Yaskawa INFORM job: KRIS_OTHER_WELDS.JBI

/JOB
//NAME KRIS_OTHER_WELDS
//POS
///NPOS 370,370,370,14,0,0
///TOOL 0
///POSTYPE PULSE
///PULSE
C00000=-36471,-76527,-106813,19264,71481,77238
C00001=-104392,-45604,-45068,-41730,67848,-43971
C00002=-102772,-23592,-15673,-48581,65359,-41958
C00003=-103105,-4521,-1193,-48225,65783,-42370
C00004=-103550,-365,5452,-48799,64222,-41754
C00005=-103550,625,8518,-49296,63299,-41230
C00006=-103550,355,7706,-49163,63541,-41368
C00007=-102300,1028,8270,-49380,64218,-41057
C00008=-102134,1217,8640,-49454,64220,-40967
C00009=-102487,1102,8722,-49434,63955,-41010
C00010=-101792,827,6993,-49227,64947,-41190
C00011=-100819,-958,-818,-48185,68095,-42388
C00012=-74228,-100728,-57385,-53918,72446,-30220
C00013=-60504,-146661,-111893,-16693,92041,63510
C00014=-81002,-144165,-111893,-31958,74905,63510
C00015=-99609,-128801,-101652,-29194,69226,57515
C00016=-99609,-127984,-100239,-29275,68831,57620
C00017=-99609,-128289,-100766,-29244,68978,57581
C00018=-102150,-129321,-101059,-28822,67791,56859
C00019=-99944,-132310,-102446,-29373,67957,57721
C00020=-94854,-157221,-110079,-32013,62771,61374
C00021=-94854,-157221,-110079,-32013,62771,61374
C00022=-150575,-180894,-113467,20602,37776,-7473
C00023=-131435,-154210,-106652,7413,43941,3112
C00024=-131414,-154056,-106648,7392,44016,3129
C00025=-131048,-150684,-105922,7028,45259,3400
C00026=-131414,-154056,-106648,7392,44016,3129
C00027=-178670,-106537,-94441,32173,86364,-27351
C00028=-174579,-86120,-85943,32864,94727,-28981
C00029=-173469,-85635,-85233,32803,94141,-28710
C00030=-173469,-85539,-84108,32766,93596,-28870
C00031=-173084,-86046,-85408,32780,93905,-28625
C00032=-171779,-87936,-86208,32689,92999,-28371
C00033=-172551,-86827,-85740,32743,93534,-28522
C00034=-185237,-110424,-94728,32531,92831,-33795
C00035=-185237,-110424,-94728,32531,92831,-33795
C00036=-134012,-175619,-118342,-2096,46955,2797
C00037=-133371,-126486,-107062,-2327,67886,2658
C00038=-134292,-123400,-104700,-2048,67993,2322
C00039=-134292,-122480,-102592,-2060,67168,2335
C00040=-134292,-122828,-103379,-2055,67474,2331
C00041=-133740,-117277,-101631,-2195,69264,2498
C00042=-134292,-122828,-103379,-2055,67474,2331
C00043=-145565,-124760,-104669,1363,67226,-1769
C00044=-155916,-134756,-102618,15305,54723,-11432
C00045=-154931,-135462,-102806,14939,54301,-11078
C00046=-159722,-139649,-104449,17130,54142,-13140
C00047=-121501,-151260,-116369,-16790,67529,22254
C00048=-84851,-125920,-106326,-14509,72614,18670
C00049=-87302,-113526,-101119,-13757,75261,17475
C00050=-88050,-112106,-100360,-13572,75391,17193
C00051=-88050,-111725,-99039,-13608,74790,17261
C00052=-88050,-111984,-99928,-13584,75193,17215
C00053=-88832,-108808,-98834,-13352,75998,16846
C00054=-87807,-112947,-100252,-13656,74947,17329
C00055=-92070,-142291,-103311,-16392,49176,14760
C00056=-92668,-139554,-102636,-15878,50013,14349
C00057=-91121,-138706,-102421,-16531,50612,14939
C00058=-93561,-140381,-102567,-15560,49394,14049
C00059=-69173,-195704,-118009,-34153,38892,29324
C00060=-69173,-195704,-118009,-34153,38892,29324
C00061=-107696,-37154,-67359,-5229,84713,5863
C00062=-116742,-32674,-55171,-12076,80004,1616
C00063=-117154,-30403,-53709,-11929,80206,1458
C00064=-117154,-30689,-52627,-11956,79411,1536
C00065=-117154,-30552,-53163,-11943,79803,1497
C00066=-108517,-16990,-43540,-23191,88993,13455
C00067=-109765,-14828,-41918,-22897,88763,13064
C00068=-109347,-17906,-44920,-22997,89117,13141
C00069=-106896,-6499,-37008,-27511,96493,19470
C00070=-107863,-6880,-37313,-27352,96184,19193
C00071=-104662,-5505,-36210,-27871,97208,20107
C00072=-93389,-55640,-71668,-19302,82770,9184
C00073=-93389,-55640,-71668,-19302,92834,-78584
C00074=-111754,-46764,-69921,-16160,92456,-84768
C00075=-113010,-47490,-70150,-15902,91999,-85126
C00076=-113010,-47824,-69220,-15892,91281,-85034
C00077=-113010,-47731,-69491,-15895,91487,-85061
C00078=-112902,-49890,-70751,-15912,91185,-84985
C00079=-100788,-44242,-62951,-32464,93570,-83345
C00080=-95750,-41506,-57227,-39958,94516,-82624
C00081=-97351,-42547,-57870,-39748,93692,-82997
C00082=-107713,-44703,-69881,-16984,94226,-83661
C00083=-110462,-17925,-52010,-16025,110800,-86473
C00084=-113105,-11726,-45581,-15485,114570,-87767
C00085=-116727,-11513,-45414,-15662,113935,-88992
C00086=-102039,-2481,-42089,-15122,118996,-84328
C00087=-102039,-2481,-42089,-15122,100704,14672
C00088=-117847,-25402,-50017,-12117,83012,11069
C00089=-117859,-24620,-49869,-12107,83315,11036
C00090=-117859,-24721,-49537,-12111,83065,11060
C00091=-117448,-24507,-49386,-12236,83141,11189
C00092=-109902,-9247,-38011,-19141,88596,18895
C00093=-104609,19012,-13716,-27585,102398,34238
C00094=-104836,21780,-11197,-27552,102213,34199
C00095=-98934,25941,-685,-39115,101412,35075
C00096=-91600,14785,-13342,-39748,106246,36411
C00097=-47111,-89064,-83881,-31350,116876,52529
C00098=-81588,-140072,-114826,-15376,71241,20037
C00099=-97769,-116268,-100554,-7249,70146,8698
C00100=-93709,-113858,-99760,-8341,71283,10082
C00101=-110362,-115244,-100357,6076,70211,-7492
C00102=-124823,-97243,-93907,17727,83078,-24095
C00103=-122674,-104476,-96562,17426,80631,-23684
C00104=-131812,-116317,-102091,19024,80117,-27039
C00105=-131812,-116317,-102091,19024,80117,-27039
C00106=-106372,-151670,-115941,-1479,61909,1124
C00107=-97402,-154853,-108420,-9880,47553,8329
C00108=-91237,-150897,-107478,-16251,51513,16477
C00109=-91228,-148864,-107179,-20465,55021,21052
C00110=-78071,-160284,-116606,-19433,65818,26969
C00111=-78071,-160284,-116606,-19433,65818,26969
C00112=-90794,-133617,-109168,-16116,71767,21274
C00113=-91693,-124585,-104857,-15775,73503,20713
C00114=-94506,-128481,-105877,-15295,71639,19928
C00115=-115362,-143961,-110168,-10698,63087,13119
C00116=-118733,-159504,-110501,-11315,48800,13248
C00117=-120726,-159269,-110393,-10449,48589,12395
C00118=-145117,-154970,-109769,815,48979,1768
C00119=-160284,-149983,-108729,14151,53864,-11283
C00120=-160335,-149941,-108719,14167,53888,-11301
C00121=-182605,-105442,-95794,27625,86766,-32303
C00122=-182041,-70442,-81142,28906,106085,-40460
C00123=-180373,-64217,-77967,29369,107732,-40648
C00124=-198406,-78013,-87317,27723,112552,-46613
C00125=-172769,-133105,-108161,-8035,62165,26522
C00126=-178553,-109735,-99654,4570,64842,24680
C00127=-178553,-100066,-94046,4517,66355,24740
C00128=-175583,-95072,-92228,3296,67653,25861
C00129=-192352,-138021,-108691,10814,57252,18824
C00130=-195651,-141887,-109704,12316,56387,17389
C00131=-195651,-141887,-109704,12316,56387,17389
C00132=-147222,-76033,-86464,-7641,74662,35625
C00133=-144580,-61393,-75556,-8586,75722,36452
C00134=-156265,-37930,-66612,3030,87434,69848
C00135=-155034,-33755,-60965,2668,86065,70206
C00136=-154458,-32798,-60008,2135,86746,70342
C00137=-155825,-31413,-58479,2524,86554,69904
C00138=-162790,-57725,-64353,16754,59169,66258
C00139=-162790,-57725,-64353,16754,59169,66258
C00140=-155825,-31413,-58479,2524,86554,69904
C00141=-155825,-31413,-58479,2524,86554,69904
C00142=-162790,-57725,-64353,16754,59169,66258
C00143=-165729,-66356,-73131,18164,60713,65340
C00144=-165729,-63659,-85226,16965,69151,66660
C00145=-19938,-154159,-115231,23119,85461,7967
C00146=-13636,-159467,-113845,12203,49637,17715
C00147=-116484,-130017,-129030,11526,91164,19547
C00148=-116484,-130017,-129030,11526,91164,19547
C00149=-101509,-111741,-97351,-2474,75173,11228
C00150=-109604,-105261,-90247,-737,73969,8417
C00151=-109604,-104665,-88539,-738,73224,8421
C00152=-109604,-104936,-89303,-737,73555,8419
C00153=-110002,-100393,-87649,-645,74866,8273
C00154=-109618,-105123,-90216,-732,74019,8412
C00155=-74185,-80593,-80392,-7895,82492,20315
C00156=-74487,-79761,-79527,-7841,82359,20221
C00157=-74487,-79638,-78308,-7850,81677,20261
C00158=-74487,-79693,-78808,-7845,81955,20243
C00159=-75396,-77288,-77713,-7667,82425,19905
C00160=-74164,-80634,-80212,-7899,82363,20329
C00161=-71363,-97810,-96211,-8399,83653,21197
C00162=-71363,-97810,-96211,-8399,83653,21197
C00163=-75126,-80656,-81685,-7709,83157,19951
C00164=-76229,-77543,-78801,-7504,82880,19595
C00165=-76229,-77418,-77195,-7514,81965,19651
C00166=-76229,-77461,-77677,-7510,82237,19634
C00167=-77485,-73926,-76028,-7263,82920,19167
C00168=-76229,-77506,-78245,-7506,82561,19615
C00169=-111141,-100889,-88631,-397,75213,7875
C00170=-111199,-100043,-88075,-385,75306,7854
C00171=-111199,-99510,-86287,-385,74481,7854
C00172=-111199,-99854,-87425,-384,75005,7852
C00173=-111556,-94962,-85553,-305,76365,7724
C00174=-110981,-102889,-89081,-432,74466,7929
C00175=-63222,-84337,-117253,-10216,104159,22323
C00176=-63222,-84337,-117253,-10216,104159,22323
C00177=-116461,-126066,-89110,816,62587,5937
C00178=-121112,-11531,-1732,22241,71063,-6555
C00179=-123069,21697,30953,28709,69461,-10931
C00180=-122369,24261,34644,28789,68382,-10931
C00181=-122349,25171,36872,28955,67580,-11137
C00182=-124729,43924,54800,30715,75908,-19671
C00183=-123229,45725,56700,30654,75959,-19910
C00184=-122369,24261,34644,28789,68382,-10931
C00185=-122757,31247,42135,29026,67616,-11292
C00186=-122369,32445,43348,29004,67370,-11200
C00187=-122776,30953,41451,28977,67860,-11234
C00188=-124792,19441,29060,28915,70056,-11467
C00189=-123719,29254,39551,29128,68728,-50133
C00190=-123432,29487,40138,29139,68416,-50100
C00191=-123432,30301,42102,29286,67723,-50287
C00192=-123432,29794,40884,29194,68152,-50171
C00193=-122305,29700,40790,29062,67775,-49816
C00194=-123432,29794,40884,29194,68152,-50171
C00195=-130745,-67077,-33050,30688,66975,-53477
C00196=-125856,-63248,-28818,30456,64700,-52130
C00197=-125856,-62207,-26795,30622,64084,-52309
C00198=-125856,-62769,-27883,30532,64415,-52213
C00199=-123740,-62907,-27951,30347,63650,-51561
C00200=-125856,-63248,-28818,30456,64700,-52130
C00201=-154464,-88255,-48627,31084,74327,-60840
C00202=-106362,-64202,-67111,-7532,73191,21872
C00203=-94843,-131680,-92775,-12823,56012,27739
C00204=-140364,-112792,-85989,36793,59691,67841
C00205=-158545,-73764,-60782,39609,71363,63907
C00206=-158545,-73538,-60068,39675,71111,63809
C00207=-158220,-67471,-54290,39710,70623,63764
C00208=-158220,-67064,-53033,39832,70183,63590
C00209=-158220,-67225,-53525,39784,70354,63658
C00210=-159834,-65842,-52837,39997,71318,63299
C00211=-159834,-65842,-52837,39997,71318,63299
C00212=-159366,-66137,-52690,39970,70914,63355
C00213=-160474,-67684,-54367,40105,71611,63123
C00214=-187581,-124736,-92952,42921,80369,54295
C00215=-106362,-64202,-67111,-7532,73191,21872
C00216=-114111,-33769,-47951,-4944,76427,19032
C00217=-116170,-28158,-40224,-4312,74444,18403
C00218=-116170,-28142,-38824,-4327,73592,18433
C00219=-116170,-28153,-39295,-4321,73875,18423
C00220=-116253,-25293,-37304,-4290,74115,18387
C00221=-114317,-34919,-41800,-5611,66541,19356
C00222=-114260,-33378,-40787,-5626,66711,19367
C00223=-115034,-33499,-40868,-5308,66647,19089
C00224=-113158,-36981,-44175,-6067,67023,19752
C00225=-112664,-46710,-50923,-6306,66218,19974
C00226=-89680,-35115,-43687,-15042,70735,27919
C00227=-91637,-21855,-35421,-13091,75116,26782
C00228=-91876,-20585,-33111,-13073,74332,26785
C00229=-91876,-20566,-32258,-13104,73831,26840
C00230=-91876,-20585,-33111,-13073,74332,26785
C00231=-92389,-17919,-31150,-12899,74409,26598
C00232=-92130,-19322,-32180,-12987,74366,26692
C00233=-94093,-21573,-33801,-12367,73907,26048
C00234=-94752,-22029,-34122,-12156,73773,25827
C00235=-94116,-21556,-33780,-12360,73899,26041
C00236=-89471,-44398,-62631,-13554,80495,26944
C00237=-122819,-38731,-49409,-10163,73779,23755
C00238=-123901,-31517,-41329,-9859,72397,23490
C00239=-123898,-31367,-41229,-9859,72412,23490
C00240=-123846,-28795,-39484,-9864,72664,23488
C00241=-122861,-32799,-42184,-10217,72396,23858
C00242=-117239,-31881,-41533,-12078,73231,25771
C00243=-117050,-26971,-37987,-12120,73592,25801
C00244=-117050,-26927,-36697,-12165,72838,25879
C00245=-118428,-26989,-37557,-11688,73120,25361
C00246=-119059,-27021,-37582,-11480,73027,25151
C00247=-118425,-26908,-37435,-11691,73088,25365
C00248=-118304,-35951,-45306,-11721,73299,25387
C00249=-123411,-39440,-45986,27831,73569,-1045
C00250=-123203,-26968,-33658,27929,72456,-1240
C00251=-123203,-26817,-32292,28037,71780,-1409
C00252=-123203,-26931,-33292,27958,72274,-1285
C00253=-123173,-25001,-31943,27927,72407,-1239
C00254=-123137,-22619,-30252,27893,72558,-1186
C00255=-123207,-27107,-33414,27962,72262,-1288
C00256=-122069,-27891,-33955,27643,71824,-948
C00257=-121286,-27911,-33965,27413,71565,-701
C00258=-122261,-27884,-33947,27698,71888,-1006
C00259=-122377,-39377,-48800,27318,74811,-339
C00260=-122377,-39377,-48800,15958,74811,-37256
C00261=-116853,-24659,-37061,14175,74133,-35375
C00262=-116391,-23304,-34381,14087,73131,-35328
C00263=-116890,-18023,-30542,14224,73560,-35454
C00264=-117861,-38592,-48080,14522,73947,-35755
C00265=-104583,-32490,-50397,-7546,82362,-7604
C00266=-105194,-26999,-38249,-8695,72546,-7274
C00267=-106425,-25461,-35908,-8300,71776,-7651
C00268=-105621,-25344,-35679,-8584,71778,-7370
C00269=-94756,-24495,-35182,-12212,73294,-3657
C00270=-93464,-24093,-34911,-12626,73531,-3224
C00271=-84425,-15663,-28771,-15378,75611,-260
C00272=-84409,-15646,-28758,-15383,75615,-255
C00273=-74667,15852,-2472,-27743,93804,20413
C00274=-73176,33846,16200,-30169,99857,32258
C00275=-73175,34349,17285,-31271,97906,32705
C00276=-67749,23419,3523,-31459,102357,33616
C00277=-95915,-30118,-44789,-16449,81748,17699
C00278=-99498,-19735,-34684,-15585,80206,16655
C00279=-100845,-17231,-31009,-15280,79016,16337
C00280=-102137,-19734,-32785,-12692,77192,13189
C00281=-98777,-17805,-31354,-13619,77838,14290
C00282=-114046,-21233,-33889,8190,75173,-9262
C00283=-113751,-21180,-33859,8096,75154,-9161
C00284=-113262,-31754,-46716,7868,77565,-8837
C00285=-121052,-35480,-50751,-8872,78740,8774
C00286=-126219,-34781,-43956,-7407,74440,7288
C00287=-119196,-19919,-32948,-16697,80290,18377
C00288=-118888,-19189,-32414,-16769,80395,18472
C00289=-117843,-14611,-28954,-17006,80823,18778
C00290=-126194,-23545,-35533,-5625,74578,5335
C00291=-131876,-24273,-36050,2510,74039,-3301
C00292=-129512,-24976,-36546,1741,73923,-2487
C00293=-130676,-43988,-54039,2112,74946,-2871
C00294=-144327,-162746,-116257,7792,53093,-8922
C00295=-140364,-112792,-85989,36793,59691,67841
C00296=-158545,-73764,-60782,39609,71363,63907
C00297=-154861,-52064,-52586,29243,83996,69304
C00298=-154351,-49821,-50803,28581,84911,69703
C00299=-152503,-51218,-50855,28383,83675,70107
C00300=-163830,-77249,-47217,57437,56476,52886
C00301=-164600,-79193,-48735,57564,56899,52688
C00302=-152503,-51284,-51279,28373,83875,70156
C00303=-152503,-51218,-50855,28383,83675,70107
C00304=-163830,-77249,-47217,57437,56476,52886
C00305=-164600,-79193,-48735,57564,56899,52688
C00306=-211845,-135273,-82829,57573,80898,40537
C00307=-8980,-110764,-82837,4940,58692,-5944
C00308=-63222,-84337,-117253,-10216,104159,22323
C00309=-63222,-84337,-117253,-10216,104159,22323
C00310=-62622,-35658,-60172,-17305,99584,35384
C00311=-67983,-29131,-50691,-16571,96143,34035
C00312=-68331,-28501,-48838,-16498,95293,34032
C00313=-95632,-58371,-67003,-12438,86482,25776
C00314=-93243,-56160,-71235,-12854,90500,26173
C00315=-74215,-69707,-85545,-7852,91184,19756
C00316=-93841,-69746,-85565,9172,91908,-7615
C00317=-97380,-51119,-65343,9768,89472,-8971
C00318=-98327,-45227,-60309,9943,89518,-9282
C00319=-98294,-45060,-62789,9947,91102,-9145
C00320=-97224,-52262,-64508,9752,88371,-9004
C00321=-70381,-14792,-39425,4699,89806,-65
C00322=-72305,-19661,-49372,5108,93524,-541
C00323=-103604,-85812,-120886,11405,106313,-9533
C00324=-4313,-85812,-120886,11405,106313,-9533
C00325=-4313,-85812,-120886,11405,106313,-9533
C00326=-116461,-126066,-89110,816,62587,5937
C00327=-120494,-28298,-18223,19234,72094,-4641
C00328=-115081,317,11412,13994,56205,-7379
C00329=-111973,8932,21807,13104,53769,-6409
C00330=-111881,7001,20107,13059,53806,-6365
C00331=-111973,8122,19702,12964,54626,-6300
C00332=-115099,15392,27643,14375,54029,-7689
C00333=-123046,33928,45673,26890,63674,-23672
C00334=-126089,67374,82990,30684,71048,-36378
C00335=-126005,74918,92279,31006,69428,-36805
C00336=-129411,35206,44111,29718,78661,-35512
C00337=-130589,8419,18518,29555,80810,-75073
C00338=-123809,36648,48124,26197,90527,-76461
C00339=-120323,36450,47917,26778,89457,-75412
C00340=-128053,46953,52473,25525,94200,-77226
C00341=-132423,-27016,-13437,24037,82468,-48912
C00342=-125265,-65617,-33465,24620,73519,-48112
C00343=-119803,-68649,-32776,24630,68538,-45055
C00344=-120043,-4148,7612,23637,76204,-43532
C00345=-120137,-2207,9677,23667,75980,-43615
C00346=-120228,48774,58665,24092,72379,-44394
C00347=-117419,29997,38916,19795,65734,-32891
C00348=-123699,9685,13287,20232,72289,-34129
C00349=-136612,-39302,-26410,22131,74933,-38485
C00350=-171363,-111780,-58290,25542,68690,-52860
C00351=-105993,-174005,-130935,24309,80821,-50388
C00352=-106047,-157383,-132399,-4283,59082,17249
C00353=-106047,-157383,-132399,-4283,59082,17249
C00354=-88146,-87318,-79564,-5997,74851,23158
C00355=-100398,-84385,-72843,-1794,70423,11848
C00356=-101406,-83734,-72107,-1525,70285,11491
C00357=-100271,-90451,-74903,-1851,68579,11922
C00358=-100398,-85037,-75228,-1783,71555,11832
C00359=-65698,-50289,-55297,-10306,79761,23508
C00360=-61954,-58139,-63827,-11098,81445,24649
C00361=-56555,-47628,-57747,-17133,88641,29036
C00362=-60473,-40946,-49585,-16554,86317,27992
C00363=-90417,-77335,-69150,-11158,74707,18820
C00364=-88053,-87457,-77735,-11673,75122,19621
C00365=-72402,-151240,-127472,-14898,75587,25161
C00366=-72402,-151240,-127472,-14898,75587,25161
C00367=10,-151240,-127472,-4482,80219,3882
C00368=-36471,-76527,-106813,19264,71481,77238
C00369=-36471,-76527,-106813,19264,71481,77238
BC00000=295325,674563,1075170
BC00001=296662,663643,1071739
BC00002=296662,663643,1071739
BC00003=296662,663643,1071739
BC00004=296662,663643,1071739
BC00005=296662,663643,1071739
BC00006=296662,663643,1071739
BC00007=296662,663643,1071739
BC00008=296662,663643,1071739
BC00009=296661,663644,1071738
BC00010=296661,663644,1071738
BC00011=296661,663644,1071738
BC00012=296661,663644,1071738
BC00013=41438,745200,146108
BC00014=41438,783078,82859
BC00015=41438,783078,82859
BC00016=41438,783078,82859
BC00017=41438,783078,82859
BC00018=41438,783078,82859
BC00019=41438,783078,82859
BC00020=41438,783078,82859
BC00021=102416,771174,82859
BC00022=102416,771174,82859
BC00023=102416,771174,82859
BC00024=102416,771174,82859
BC00025=102416,771174,82859
BC00026=102416,771174,82859
BC00027=102416,771174,82859
BC00028=102416,771174,82857
BC00029=102416,771174,82857
BC00030=102416,771174,82857
BC00031=102416,771174,82857
BC00032=102416,771174,82857
BC00033=102416,771174,82857
BC00034=102416,771174,82857
BC00035=359114,771174,82857
BC00036=359114,771174,82857
BC00037=359114,771174,82857
BC00038=359114,771174,82857
BC00039=359114,771174,82857
BC00040=359114,771174,82857
BC00041=359114,771174,82857
BC00042=359114,771174,82857
BC00043=359114,771174,82857
BC00044=359114,771174,82857
BC00045=359114,771174,82857
BC00046=359114,771174,82857
BC00047=359114,771174,82857
BC00048=359114,771174,82857
BC00049=359114,771174,82857
BC00050=359114,771174,82857
BC00051=359114,771174,82857
BC00052=359114,771174,82857
BC00053=359114,771174,82857
BC00054=359114,771174,82857
BC00055=359114,771174,82857
BC00056=359114,771174,82857
BC00057=359114,771174,82857
BC00058=359114,771174,82857
BC00059=359114,771174,82857
BC00060=396097,697994,577187
BC00061=396097,697994,759870
BC00062=396097,697994,759870
BC00063=396097,697994,759870
BC00064=396097,697994,759870
BC00065=396097,697994,759870
BC00066=396097,697994,759870
BC00067=396097,697994,759870
BC00068=396097,697994,759870
BC00069=396097,697994,759870
BC00070=396097,697994,759870
BC00071=396097,697994,759870
BC00072=396097,697994,759870
BC00073=396097,697994,759870
BC00074=396097,697994,759870
BC00075=396097,697994,759870
BC00076=396097,697994,759870
BC00077=396097,697994,759870
BC00078=396097,697994,759870
BC00079=396097,697994,759870
BC00080=396097,697994,759870
BC00081=396097,697994,759870
BC00082=396097,697994,759870
BC00083=396097,697995,759869
BC00084=396097,697995,759869
BC00085=396097,697995,759869
BC00086=396097,697995,759869
BC00087=396097,697995,759869
BC00088=396097,697995,759869
BC00089=396097,697995,759869
BC00090=396097,697995,759869
BC00091=396097,697995,759869
BC00092=396097,697995,759869
BC00093=396097,697995,759869
BC00094=396097,697995,759869
BC00095=396097,697995,759869
BC00096=396097,697995,759869
BC00097=396097,697995,759869
BC00098=359114,771174,82857
BC00099=359114,771174,82857
BC00100=359114,771174,82857
BC00101=359114,771174,82857
BC00102=359114,771174,82857
BC00103=359114,771174,82857
BC00104=359114,771174,82857
BC00105=308698,771174,82857
BC00106=314110,781864,75319
BC00107=314855,783332,74282
BC00108=314854,783334,74282
BC00109=314854,783334,74282
BC00110=314854,783334,74282
BC00111=121885,783334,74282
BC00112=121885,783334,74282
BC00113=121885,783334,74282
BC00114=121885,783334,74282
BC00115=121885,783334,74282
BC00116=121885,783334,74282
BC00117=121885,783334,74282
BC00118=121885,783334,74282
BC00119=121885,783334,74282
BC00120=121885,783334,74282
BC00121=121885,783334,74282
BC00122=121885,783334,74282
BC00123=121885,783334,74282
BC00124=121885,783334,74282
BC00125=121885,783334,74282
BC00126=121885,783334,74282
BC00127=121885,783334,74282
BC00128=121885,783334,74282
BC00129=121885,783334,74282
BC00130=269139,680260,222960
BC00131=368841,723129,895975
BC00132=368840,723129,895974
BC00133=368840,723129,895974
BC00134=368840,723129,895974
BC00135=368840,723129,895974
BC00136=368840,723129,895974
BC00137=368840,723129,895974
BC00138=368840,723129,895974
BC00139=368840,723129,900139
BC00140=368840,723129,902099
BC00141=368840,723129,895974
BC00142=368840,723129,895974
BC00143=368840,723129,895974
BC00144=368840,723129,895974
BC00145=323544,666412,663921
BC00146=215473,679246,1035002
BC00147=215473,679246,1061707
BC00148=302549,801305,1061707
BC00149=302549,801305,1022507
BC00150=302549,801305,1022507
BC00151=302549,801305,1022507
BC00152=302549,801305,1022507
BC00153=302549,801305,1022507
BC00154=302549,801305,1022507
BC00155=302549,801305,1022507
BC00156=302549,801305,1022507
BC00157=302549,801305,1022507
BC00158=302549,801305,1022507
BC00159=302549,801305,1022507
BC00160=302549,801305,1022507
BC00161=291909,797081,1023585
BC00162=48431,797081,1023585
BC00163=48431,797081,1023585
BC00164=48431,797081,1023585
BC00165=48431,797081,1023585
BC00166=48431,797081,1023585
BC00167=48431,797081,1023585
BC00168=48431,797081,1023585
BC00169=48431,797081,1023585
BC00170=48431,797081,1023585
BC00171=48431,797081,1023585
BC00172=48431,797081,1023585
BC00173=48431,797081,1023585
BC00174=48431,797081,1023585
BC00175=48431,797081,1023585
BC00176=21691,673150,1023585
BC00177=2007,673150,1023585
BC00178=2008,673150,1023583
BC00179=2008,673150,1023582
BC00180=2008,673150,1023582
BC00181=2008,673150,1023582
BC00182=2008,673150,1023582
BC00183=2008,673150,1023582
BC00184=2008,673150,1023582
BC00185=2008,673150,1023582
BC00186=2008,673150,1023582
BC00187=2008,673150,1023582
BC00188=2008,673150,1023582
BC00189=2008,673150,1023579
BC00190=2008,673150,1023579
BC00191=2008,673150,1023579
BC00192=2008,673150,1023579
BC00193=2008,673150,1023579
BC00194=2008,673150,1023579
BC00195=2008,673150,1023579
BC00196=2008,673150,1023579
BC00197=2008,673150,1023579
BC00198=2008,673150,1023579
BC00199=2008,673150,1023579
BC00200=2008,673150,1023579
BC00201=2008,673150,1023579
BC00202=48431,687657,196518
BC00203=170480,697437,1002568
BC00204=170479,738837,1002567
BC00205=170479,738837,1002567
BC00206=170479,738837,1002567
BC00207=170479,738837,1002567
BC00208=170479,738837,1002567
BC00209=170479,738837,1002567
BC00210=170479,738837,1002567
BC00211=170479,738837,1002567
BC00212=170479,738837,1002567
BC00213=170479,738837,1002567
BC00214=170479,738837,1002567
BC00215=48431,687657,196518
BC00216=48431,687657,196518
BC00217=48431,687657,196518
BC00218=48431,687657,196518
BC00219=48431,687657,196518
BC00220=48431,687657,196518
BC00221=48431,687657,196518
BC00222=48431,687657,196518
BC00223=48431,687657,196518
BC00224=48431,687657,196518
BC00225=48431,687657,196518
BC00226=48431,687657,196518
BC00227=48431,687657,196518
BC00228=48431,687657,196516
BC00229=48431,687657,196516
BC00230=48431,687657,196516
BC00231=48431,687657,196516
BC00232=48431,687657,196516
BC00233=48431,687657,196516
BC00234=48431,687657,196516
BC00235=48431,687657,196516
BC00236=48431,687657,196516
BC00237=376831,687657,196515
BC00238=376831,687657,196515
BC00239=376831,687657,196515
BC00240=376831,687657,196515
BC00241=376831,687657,196515
BC00242=376831,687657,196515
BC00243=376831,687657,196515
BC00244=376831,687657,196515
BC00245=376831,687657,196515
BC00246=376831,687657,196515
BC00247=376831,687657,196515
BC00248=376831,687657,196515
BC00249=376831,687657,196515
BC00250=376831,687657,196515
BC00251=376831,687657,196515
BC00252=376831,687657,196515
BC00253=376831,687657,196515
BC00254=376831,687657,196515
BC00255=376831,687657,196515
BC00256=376831,687657,196515
BC00257=376831,687657,196515
BC00258=376831,687657,196515
BC00259=376831,687657,196515
BC00260=376831,687657,196515
BC00261=376831,687657,196513
BC00262=376831,687657,196513
BC00263=376831,687657,196513
BC00264=376831,687657,196513
BC00265=271972,687657,196507
BC00266=271972,687657,196507
BC00267=271972,687657,196507
BC00268=271972,687657,196507
BC00269=271972,687657,196507
BC00270=271972,687657,196507
BC00271=271972,687657,196507
BC00272=271972,687657,196507
BC00273=271972,687657,196507
BC00274=271972,687657,196507
BC00275=271972,687657,196507
BC00276=271972,687657,196507
BC00277=72168,687657,196500
BC00278=72168,687657,196500
BC00279=72168,687657,196498
BC00280=72168,687657,196498
BC00281=72168,687657,196498
BC00282=72168,687657,196496
BC00283=72168,687657,196496
BC00284=72168,687657,196496
BC00285=72168,687657,196499
BC00286=72169,687657,196497
BC00287=72169,687657,196497
BC00288=72169,687657,196497
BC00289=72169,687657,196497
BC00290=72169,687657,196497
BC00291=72169,687657,196497
BC00292=72169,687657,196497
BC00293=72169,687657,196497
BC00294=130997,687657,956487
BC00295=170479,738837,1002567
BC00296=170479,738837,1002567
BC00297=170479,738837,1002567
BC00298=170479,738837,1002567
BC00299=170479,738837,1002567
BC00300=170479,738837,1002567
BC00301=170479,738837,1002567
BC00302=170479,738837,1002567
BC00303=170479,738837,1002567
BC00304=170479,738837,1002567
BC00305=170479,738837,1002567
BC00306=170479,738837,1002567
BC00307=72169,665569,501851
BC00308=21691,673150,1023585
BC00309=31859,773328,1023585
BC00310=31859,773328,1023580
BC00311=31859,773328,1023580
BC00312=31859,773328,1023577
BC00313=31858,773328,1023571
BC00314=31858,773328,1023571
BC00315=31859,773328,1023585
BC00316=239094,773328,1023585
BC00317=239094,773328,1023585
BC00318=239094,773328,1023583
BC00319=239094,773328,1023583
BC00320=239094,773328,1023583
BC00321=239094,773328,1023583
BC00322=239094,773328,1023583
BC00323=239094,773328,1023583
BC00324=178929,686286,1023583
BC00325=46757,686286,1023583
BC00326=2007,673150,1023585
BC00327=2008,673151,1023581
BC00328=2009,673152,1023573
BC00329=2009,673152,1023573
BC00330=2009,673152,1023573
BC00331=2009,673152,1023573
BC00332=2009,673152,1023573
BC00333=2009,673152,1023573
BC00334=2009,673152,1023573
BC00335=2009,673152,1023573
BC00336=2009,673152,1023573
BC00337=2009,673152,1023573
BC00338=2009,673152,1023573
BC00339=2009,673152,1023573
BC00340=2009,673152,1023573
BC00341=2009,673152,1023573
BC00342=2009,673152,1023573
BC00343=2009,673152,1023573
BC00344=2009,673152,1023573
BC00345=2009,673152,1023573
BC00346=2009,673152,1023573
BC00347=2009,673152,1023573
BC00348=2009,673152,1023573
BC00349=2009,673152,1023573
BC00350=2009,679183,1023573
BC00351=2009,719980,1066462
BC00352=2009,719980,1066462
BC00353=84626,785651,1066462
BC00354=84626,785651,1066462
BC00355=84626,785651,1066462
BC00356=84626,785651,1066462
BC00357=84626,785651,1066462
BC00358=84626,785651,1066462
BC00359=84626,785651,1066462
BC00360=84626,785651,1066462
BC00361=211931,785651,1066462
BC00362=211931,785651,1066462
BC00363=211931,785651,1066462
BC00364=211931,785651,1066462
BC00365=211931,792271,1066462
BC00366=211931,702469,1066462
BC00367=211931,670537,1065237
BC00368=295325,674563,1075170
BC00369=295325,674563,1075170
EC00000=-1596315,0
EC00001=-1596315,0
EC00002=-1596315,0
EC00003=-1596315,0
EC00004=-1596315,0
EC00005=-1596315,0
EC00006=-1596315,0
EC00007=-1596315,0
EC00008=-1596315,0
EC00009=-1596315,0
EC00010=-1596315,0
EC00011=-1596315,0
EC00012=-1596315,0
EC00013=-1596315,0
EC00014=-1596315,0
EC00015=-1596315,0
EC00016=-1596315,0
EC00017=-1596315,0
EC00018=-1596315,0
EC00019=-1596315,0
EC00020=-1596315,0
EC00021=-1596315,0
EC00022=-1596315,0
EC00023=-1596315,0
EC00024=-1596315,0
EC00025=-1596315,0
EC00026=-1596315,0
EC00027=-1596315,0
EC00028=-1596315,0
EC00029=-1596315,0
EC00030=-1596315,0
EC00031=-1596315,0
EC00032=-1596315,0
EC00033=-1596315,0
EC00034=-1596315,0
EC00035=-1596315,0
EC00036=-1596315,0
EC00037=-1596315,0
EC00038=-1596315,0
EC00039=-1596315,0
EC00040=-1596315,0
EC00041=-1596315,0
EC00042=-1596315,0
EC00043=-1596315,0
EC00044=-1596315,0
EC00045=-1596315,0
EC00046=-1596315,0
EC00047=-1596315,0
EC00048=-1596315,0
EC00049=-1596315,0
EC00050=-1596315,0
EC00051=-1596315,0
EC00052=-1596315,0
EC00053=-1596315,0
EC00054=-1596315,0
EC00055=-1596315,0
EC00056=-1596315,0
EC00057=-1596315,0
EC00058=-1596315,0
EC00059=-1596315,0
EC00060=-1596315,0
EC00061=-1863244,-545567
EC00062=-1863244,-545567
EC00063=-1863244,-545567
EC00064=-1863244,-545567
EC00065=-1863244,-545567
EC00066=-1863244,-545567
EC00067=-1863244,-545567
EC00068=-1863244,-545567
EC00069=-1863244,-545567
EC00070=-1863244,-545567
EC00071=-1863244,-545567
EC00072=-1863244,-545567
EC00073=-1863244,-545567
EC00074=-1863244,-545567
EC00075=-1863244,-545567
EC00076=-1863244,-545567
EC00077=-1863244,-545567
EC00078=-1863244,-545567
EC00079=-1863244,-545567
EC00080=-1863244,-545567
EC00081=-1863244,-545567
EC00082=-1863244,-545567
EC00083=-1863245,-545566
EC00084=-1863246,-545566
EC00085=-1863246,-545566
EC00086=-1863246,-545566
EC00087=-1863246,-545566
EC00088=-1863246,-545566
EC00089=-1863246,-545566
EC00090=-1863246,-545566
EC00091=-1863246,-545566
EC00092=-1863246,-545566
EC00093=-1863246,-545566
EC00094=-1863246,-545566
EC00095=-1863246,-545566
EC00096=-1863246,-545566
EC00097=-1863246,-545566
EC00098=-1596315,0
EC00099=-1596315,0
EC00100=-1596315,0
EC00101=-1596315,0
EC00102=-1596315,0
EC00103=-1596315,0
EC00104=-1596315,0
EC00105=-1596315,0
EC00106=-1596315,0
EC00107=-1596315,0
EC00108=-1596315,0
EC00109=-1596315,0
EC00110=-1596315,0
EC00111=-1596315,0
EC00112=-1596315,0
EC00113=-1596315,0
EC00114=-1596315,0
EC00115=-1596315,0
EC00116=-1596315,0
EC00117=-1596315,0
EC00118=-1596315,0
EC00119=-1596315,0
EC00120=-1596315,0
EC00121=-1596315,0
EC00122=-1596315,0
EC00123=-1596315,0
EC00124=-1596315,0
EC00125=-1596315,0
EC00126=-1596315,0
EC00127=-1596315,0
EC00128=-1596315,0
EC00129=-1596315,0
EC00130=-1596315,0
EC00131=-1596315,0
EC00132=-1596317,0
EC00133=-1596317,0
EC00134=-1596317,0
EC00135=-1596317,0
EC00136=-1596317,0
EC00137=-1596317,0
EC00138=-1596317,0
EC00139=-1596317,0
EC00140=-1596317,0
EC00141=-1596317,0
EC00142=-1596317,0
EC00143=-1596317,0
EC00144=-1596317,0
EC00145=-1596882,-556476
EC00146=-1857823,-556476
EC00147=-1857823,-556476
EC00148=-1857823,-556476
EC00149=-1857823,-556476
EC00150=-1857823,-556476
EC00151=-1857823,-556476
EC00152=-1857823,-556476
EC00153=-1857823,-556476
EC00154=-1857823,-556476
EC00155=-1857823,-556476
EC00156=-1857823,-556476
EC00157=-1857823,-556476
EC00158=-1857823,-556476
EC00159=-1857823,-556476
EC00160=-1857823,-556476
EC00161=-1857823,-556476
EC00162=-1857823,-556476
EC00163=-1857823,-556476
EC00164=-1857823,-556476
EC00165=-1857823,-556476
EC00166=-1857823,-556476
EC00167=-1857823,-556476
EC00168=-1857823,-556476
EC00169=-1857823,-556476
EC00170=-1857823,-556476
EC00171=-1857823,-556476
EC00172=-1857823,-556476
EC00173=-1857823,-556476
EC00174=-1857823,-556476
EC00175=-1857823,-556476
EC00176=-1857823,-556476
EC00177=-1857823,-556476
EC00178=-1857824,-556476
EC00179=-1857824,-556476
EC00180=-1857824,-556476
EC00181=-1857824,-556476
EC00182=-1857824,-556476
EC00183=-1857824,-556476
EC00184=-1857824,-556476
EC00185=-1857824,-556476
EC00186=-1857824,-556476
EC00187=-1857824,-556476
EC00188=-1857824,-556476
EC00189=-1857824,-556476
EC00190=-1857824,-556476
EC00191=-1857824,-556476
EC00192=-1857824,-556476
EC00193=-1857824,-556476
EC00194=-1857824,-556476
EC00195=-1857824,-556476
EC00196=-1857824,-556476
EC00197=-1857824,-556476
EC00198=-1857824,-556476
EC00199=-1857824,-556476
EC00200=-1857824,-556476
EC00201=-1857824,-556476
EC00202=-1596314,-1112952
EC00203=-1596314,-1112952
EC00204=-1596314,-1112951
EC00205=-1596314,-1112951
EC00206=-1596314,-1112951
EC00207=-1596314,-1112951
EC00208=-1596314,-1112951
EC00209=-1596314,-1112951
EC00210=-1596314,-1112951
EC00211=-1596314,-1112951
EC00212=-1596314,-1112951
EC00213=-1596314,-1112951
EC00214=-1596314,-1112951
EC00215=-1596314,-1112952
EC00216=-1596314,-1112952
EC00217=-1596314,-1112952
EC00218=-1596314,-1112952
EC00219=-1596314,-1112952
EC00220=-1596314,-1112952
EC00221=-1596314,-1112952
EC00222=-1596314,-1112952
EC00223=-1596314,-1112952
EC00224=-1596314,-1112952
EC00225=-1596314,-1112952
EC00226=-1596314,-1112952
EC00227=-1596314,-1112952
EC00228=-1596314,-1112951
EC00229=-1596314,-1112951
EC00230=-1596314,-1112951
EC00231=-1596314,-1112951
EC00232=-1596314,-1112951
EC00233=-1596314,-1112951
EC00234=-1596314,-1112951
EC00235=-1596314,-1112951
EC00236=-1596314,-1112951
EC00237=-1596314,-1112951
EC00238=-1596314,-1112951
EC00239=-1596314,-1112951
EC00240=-1596314,-1112951
EC00241=-1596314,-1112951
EC00242=-1596314,-1112951
EC00243=-1596314,-1112951
EC00244=-1596314,-1112951
EC00245=-1596314,-1112951
EC00246=-1596314,-1112951
EC00247=-1596314,-1112951
EC00248=-1596314,-1112951
EC00249=-1596314,-1112951
EC00250=-1596314,-1112951
EC00251=-1596314,-1112951
EC00252=-1596314,-1112951
EC00253=-1596314,-1112951
EC00254=-1596314,-1112951
EC00255=-1596314,-1112951
EC00256=-1596314,-1112951
EC00257=-1596314,-1112951
EC00258=-1596314,-1112951
EC00259=-1596314,-1112951
EC00260=-1596314,-1112951
EC00261=-1596314,-1112951
EC00262=-1596314,-1112951
EC00263=-1596314,-1112951
EC00264=-1596314,-1112951
EC00265=-1596314,-1112951
EC00266=-1596314,-1112951
EC00267=-1596314,-1112951
EC00268=-1596314,-1112951
EC00269=-1596314,-1112951
EC00270=-1596314,-1112951
EC00271=-1596314,-1112951
EC00272=-1596314,-1112951
EC00273=-1596314,-1112951
EC00274=-1596314,-1112951
EC00275=-1596314,-1112951
EC00276=-1596314,-1112951
EC00277=-1596314,-1112951
EC00278=-1596314,-1112951
EC00279=-1596314,-1112951
EC00280=-1596314,-1112951
EC00281=-1596314,-1112951
EC00282=-1596314,-1112951
EC00283=-1596314,-1112951
EC00284=-1596314,-1112951
EC00285=-1596314,-1112951
EC00286=-1596314,-1112951
EC00287=-1596314,-1112951
EC00288=-1596314,-1112951
EC00289=-1596314,-1112951
EC00290=-1596314,-1112951
EC00291=-1596314,-1112951
EC00292=-1596314,-1112951
EC00293=-1596314,-1112951
EC00294=-1596314,-1112951
EC00295=-1596314,-1112951
EC00296=-1596314,-1112951
EC00297=-1596314,-1112950
EC00298=-1596314,-1112950
EC00299=-1596314,-1112950
EC00300=-1596314,-1112950
EC00301=-1596314,-1112950
EC00302=-1596314,-1112950
EC00303=-1596314,-1112950
EC00304=-1596314,-1112950
EC00305=-1596314,-1112950
EC00306=-1596314,-1112950
EC00307=-1596314,-1112951
EC00308=-1857823,-556476
EC00309=-1857823,-556476
EC00310=-1857825,-556476
EC00311=-1857825,-556476
EC00312=-1857826,-556476
EC00313=-1857827,-556476
EC00314=-1857827,-556476
EC00315=-1857823,-556476
EC00316=-1857823,-556476
EC00317=-1857823,-556476
EC00318=-1857824,-556476
EC00319=-1857824,-556476
EC00320=-1857824,-556476
EC00321=-1857824,-556476
EC00322=-1857824,-556476
EC00323=-1857824,-556476
EC00324=-1857824,-556476
EC00325=-1857824,-556476
EC00326=-1857823,-556476
EC00327=-1857824,-556476
EC00328=-1857827,-556476
EC00329=-1857827,-556476
EC00330=-1857827,-556476
EC00331=-1857827,-556476
EC00332=-1857827,-556476
EC00333=-1857827,-556476
EC00334=-1857827,-556476
EC00335=-1857827,-556476
EC00336=-1857827,-556476
EC00337=-1857827,-556476
EC00338=-1857827,-556476
EC00339=-1857827,-556476
EC00340=-1857827,-556476
EC00341=-1857827,-556476
EC00342=-1857827,-556476
EC00343=-1857827,-556476
EC00344=-1857827,-556476
EC00345=-1857827,-556476
EC00346=-1857827,-556476
EC00347=-1857827,-556476
EC00348=-1857827,-556476
EC00349=-1857827,-556476
EC00350=-1857827,-556476
EC00351=-1857827,-556476
EC00352=-1857827,-556476
EC00353=-1857827,-556476
EC00354=-1857827,-556476
EC00355=-1857827,-556476
EC00356=-1857827,-556476
EC00357=-1857827,-556476
EC00358=-1857827,-556476
EC00359=-1857827,-556476
EC00360=-1857827,-556476
EC00361=-1857827,-556476
EC00362=-1857827,-556476
EC00363=-1857827,-556476
EC00364=-1857827,-556476
EC00365=-1857827,-556476
EC00366=-1857827,-556476
EC00367=-1857827,-556476
EC00368=-1596315,0
EC00369=0,0
///POSTYPE BASE
///RECTAN
///RCONF 0,0,0,0,0,0,0,0,0,0,0,0,0,0,0,0,0,0,0,0,0,0,0,0
P00006=0.000,0.000,0.000,0.0000,0.0000,0.0000
P00021=-0.339,1.359,3.368,0.0000,0.0000,0.0000
P00022=-0.114,-0.780,3.887,0.0000,0.0000,0.0000
P00023=0.143,-0.036,0.682,0.0000,0.0000,0.0000
P00024=0.006,-0.619,-2.354,0.0000,0.0000,0.0000
P00025=2.242,-0.049,-1.961,0.0000,0.0000,0.0000
P00026=0.572,-0.002,0.234,0.0000,0.0000,0.0000
P00027=-0.746,0.015,-9.096,0.0000,0.0000,0.0000
P00028=-2.237,-0.018,-7.702,0.0000,0.0000,0.0000
P00030=5.926,-4.294,-1.390,0.0000,0.0000,0.0000
P00031=1.853,-0.001,-1.549,0.0000,0.0000,0.0000
P00032=1.957,0.503,-7.217,0.0000,0.0000,0.0000
P00071=2.716,0.070,1.352,0.0000,0.0000,0.0000
P00072=1.041,-0.003,-0.797,0.0000,0.0000,0.0000
//INST
///DATE 2025/02/20 07:00
///ATTR SC,RW
///GROUP1 RB1,BS1
///GROUP2 ST1
NOP
MOVJ C00000 BC00000 VJ=100.00  +MOVJ EC00000 VJ=100.00
CALL JOB:CLEAN-R1_KM_NEW
MOVJ C00001 BC00001 VJ=100.00  +MOVJ EC00001 VJ=100.00
MOVJ C00002 BC00002 VJ=100.00  +MOVJ EC00002 VJ=100.00
SMOVL C00003 BC00003 V=400.0  +MOVJ EC00003
SFTOF3D
SMOVL C00004 BC00004 V=100.0  +MOVJ EC00004
SREFP 3 C00005 BC00005  +REFP EC00005
CALL JOB:SEARCH-R1-S13D
SET P071 P006
SFTON3D P071
SMOVL C00006 BC00006 V=100.0  +MOVJ EC00006
SMOVL C00007 BC00007 V=100.0  +MOVJ EC00007
SMOVL C00008 BC00008 V=83.3 PL=0  +MOVJ EC00008
SREFP 3 C00009 BC00009  +REFP EC00009
CALL JOB:SEARCH-R1-S13D
SET P071 P006
SFTON3D P071
SMOVL C00010 BC00010 V=100.0  +MOVJ EC00010
SFTOF3D
SMOVL C00011 BC00011 V=1000.0  +MOVJ EC00011
SMOVL C00012 BC00012 V=1000.0  +MOVJ EC00012
MOVJ C00013 BC00013 VJ=100.00  +MOVJ EC00013 VJ=100.00
MOVJ C00014 BC00014 VJ=100.00  +MOVJ EC00014 VJ=100.00
'SE1
SMOVL C00015 BC00015 V=100.0  +MOVJ EC00015
SREFP 3 C00016 BC00016  +REFP EC00016
CALL JOB:SEARCH-R1-S13D
SET P021 P006
SFTON3D P021
SMOVL C00017 BC00017 V=100.0  +MOVJ EC00017
SREFP 3 C00018 BC00018  +REFP EC00018
CALL JOB:SEARCH-R1-S13D
SET P021 P006
SFTON3D P021
SMOVL C00019 BC00019 V=100.0  +MOVJ EC00019
SFTOF3D
MOVJ C00020 BC00020 VJ=100.00  +MOVJ EC00020 VJ=100.00
MOVJ C00021 BC00021 VJ=100.00  +MOVJ EC00021 VJ=100.00
MOVJ C00022 BC00022 VJ=100.00  +MOVJ EC00022 VJ=100.00
MOVJ C00023 BC00023 VJ=100.00  +MOVJ EC00023 VJ=100.00
SFTOF3D
SMOVL C00024 BC00024 V=100.0  +MOVJ EC00024
SREFP 3 C00025 BC00025  +REFP EC00025
CALL JOB:SEARCH-R1-S13D
SET P022 P006
SFTON3D P022
SMOVL C00026 BC00026 V=100.0  +MOVJ EC00026
MOVJ C00027 BC00027 VJ=60.00  +MOVJ EC00027 VJ=100.00
MOVJ C00028 BC00028 VJ=60.00  +MOVJ EC00028 VJ=100.00
SMOVL C00029 BC00029 V=100.0  +MOVJ EC00029
SREFP 3 C00030 BC00030  +REFP EC00030
CALL JOB:SEARCH-R1-S13D
SET P022 P006
SFTON3D P022
SMOVL C00031 BC00031 V=100.0  +MOVJ EC00031
SREFP 3 C00032 BC00032  +REFP EC00032
CALL JOB:SEARCH-R1-S13D
SET P022 P006
SFTON3D P022
SMOVL C00033 BC00033 V=100.0  +MOVJ EC00033
SFTOF3D
'SE2
MOVJ C00034 BC00034 VJ=100.00  +MOVJ EC00034 VJ=100.00
MOVJ C00035 BC00035 VJ=100.00  +MOVJ EC00035 VJ=100.00
MOVJ C00036 BC00036 VJ=100.00  +MOVJ EC00036 VJ=100.00
MOVJ C00037 BC00037 VJ=100.00  +MOVJ EC00037 VJ=100.00
SMOVL C00038 BC00038 V=100.0  +MOVJ EC00038
SREFP 3 C00039 BC00039  +REFP EC00039
CALL JOB:SEARCH-R1-S13D
SET P023 P006
SFTON3D P023
SMOVL C00040 BC00040 V=100.0  +MOVJ EC00040
SREFP 3 C00041 BC00041  +REFP EC00041
CALL JOB:SEARCH-R1-S13D
SET P023 P006
SFTON3D P023
SMOVL C00042 BC00042 V=100.0  +MOVJ EC00042
SMOVL C00043 BC00043 V=100.0  +MOVJ EC00043
SMOVL C00044 BC00044 V=100.0  +MOVJ EC00044
SREFP 3 C00045 BC00045  +REFP EC00045
CALL JOB:SEARCH-R1-S13D
SET P023 P006
SFTON3D P023
SMOVL C00046 BC00046 V=100.0  +MOVJ EC00046
SFTOF3D
'SE3
MOVJ C00047 BC00047 VJ=100.00  +MOVJ EC00047 VJ=100.00
MOVJ C00048 BC00048 VJ=100.00  +MOVJ EC00048 VJ=100.00
MOVJ C00049 BC00049 VJ=100.00  +MOVJ EC00049 VJ=100.00
'SE4
SMOVL C00050 BC00050 V=100.0  +MOVJ EC00050
SREFP 3 C00051 BC00051  +REFP EC00051
CALL JOB:SEARCH-R1-S13D
SET P024 P006
SFTON3D P024
SMOVL C00052 BC00052 V=100.0  +MOVJ EC00052
SREFP 3 C00053 BC00053  +REFP EC00053
CALL JOB:SEARCH-R1-S13D
SET P024 P006
SFTON3D P024
SMOVL C00054 BC00054 V=100.0  +MOVJ EC00054
MOVJ C00055 BC00055 VJ=100.00  +MOVJ EC00055 VJ=100.00
SMOVL C00056 BC00056 V=100.0  +MOVJ EC00056
SREFP 3 C00057 BC00057  +REFP EC00057
CALL JOB:SEARCH-R1-S13D
SET P024 P006
SFTON3D P024
SMOVL C00058 BC00058 V=100.0  +MOVJ EC00058
SFTOF3D
MOVJ C00059 BC00059 VJ=100.00  +MOVJ EC00059 VJ=100.00
MOVJ C00060 BC00060 VJ=100.00  +MOVJ EC00060 VJ=100.00
MOVJ C00061 BC00061 VJ=100.00  +MOVJ EC00061 VJ=100.00
MOVJ C00062 BC00062 VJ=100.00  +MOVJ EC00062 VJ=100.00
'SE5
SMOVL C00063 BC00063 V=100.0  +MOVJ EC00063
SREFP 3 C00064 BC00064  +REFP EC00064
CALL JOB:SEARCH-R1-S13D
SET P025 P006
SFTON3D P025
SMOVL C00065 BC00065 V=100.0  +MOVJ EC00065
SMOVL C00066 BC00066 V=100.0  +MOVJ EC00066
SREFP 3 C00067 BC00067  +REFP EC00067
CALL JOB:SEARCH-R1-S13D
SET P025 P006
SFTON3D P025
SMOVL C00068 BC00068 V=100.0  +MOVJ EC00068
SMOVL C00069 BC00069 V=100.0  +MOVJ EC00069
SREFP 3 C00070 BC00070  +REFP EC00070
CALL JOB:SEARCH-R1-S13D
SET P025 P006
SFTON3D P025
SMOVL C00071 BC00071 V=100.0  +MOVJ EC00071
SFTOF3D
MOVJ C00072 BC00072 VJ=100.00  +MOVJ EC00072 VJ=100.00
MOVJ C00073 BC00073 VJ=100.00  +MOVJ EC00073 VJ=100.00
MOVJ C00074 BC00074 VJ=100.00  +MOVJ EC00074 VJ=100.00
'SE6
SMOVL C00075 BC00075 V=100.0  +MOVJ EC00075
SREFP 3 C00076 BC00076  +REFP EC00076
CALL JOB:SEARCH-R1-S13D
SET P026 P006
SFTON3D P026
SMOVL C00077 BC00077 V=100.0  +MOVJ EC00077
SREFP 3 C00078 BC00078  +REFP EC00078
CALL JOB:SEARCH-R1-S13D
SET P026 P006
SFTON3D P026
SMOVL C00079 BC00079 V=100.0  +MOVJ EC00079
SMOVL C00080 BC00080 V=100.0  +MOVJ EC00080
SREFP 3 C00081 BC00081  +REFP EC00081
CALL JOB:SEARCH-R1-S13D
SET P026 P006
SFTON3D P026
SMOVL C00082 BC00082 V=100.0  +MOVJ EC00082
MOVJ C00083 BC00083 VJ=15.00  +MOVJ EC00083 VJ=10.00
MACRO1 MJ#(0) ARGF14
SMOVL C00084 BC00084 V=250.0 PL=0  +MOVJ EC00084
ARCON
SWVON WEV#(66)
SMOVL C00085 BC00085 V=8.3  +MOVJ EC00085
ARCOF
SWVOF
SFTOF3D
MOVJ C00086 BC00086 VJ=30.00  +MOVJ EC00086 VJ=15.00
MOVJ C00087 BC00087 VJ=100.00  +MOVJ EC00087 VJ=100.00
MACRO1 MJ#(0) ARGF9
SFTON3D P025
SREFP 1 C00088 BC00088  +REFP EC00088
SREFP 2 C00089 BC00089  +REFP EC00089
SMOVL C00090 BC00090 V=250.0 PL=0  +MOVJ EC00090
ARCON
SWVON WEV#(68)
SMOVL C00091 BC00091 V=7.5  +MOVJ EC00091
SMOVL C00092 BC00092 V=7.5  +MOVJ EC00092
SMOVL C00093 BC00093 V=10.8  +MOVJ EC00093
SMOVL C00094 BC00094 V=10.8  +MOVJ EC00094
SMOVL C00095 BC00095 V=10.0  +MOVJ EC00095
ARCOF
SWVOF
MOVJ C00096 BC00096 VJ=100.00  +MOVJ EC00096 VJ=15.00
SFTOF3D
MOVJ C00097 BC00097 VJ=100.00  +MOVJ EC00097 VJ=100.00
MOVJ C00098 BC00098 VJ=100.00  +MOVJ EC00098 VJ=100.00
MACRO1 MJ#(0) ARGF6
SFTON3D P024
SMOVL C00099 BC00099 V=250.0  +MOVJ EC00099
ARCON
SMOVL C00100 BC00100 V=10.0  +MOVJ EC00100
SMOVL C00101 BC00101 V=12.5  +MOVJ EC00101
SMOVL C00102 BC00102 V=12.5  +MOVJ EC00102
SMOVL C00103 BC00103 V=12.5  +MOVJ EC00103
ARCOF
SFTOF3D
MOVJ C00104 BC00104 VJ=15.00  +MOVJ EC00104 VJ=15.00
MOVJ C00105 BC00105 VJ=100.00  +MOVJ EC00105 VJ=15.00
MACRO1 MJ#(0) ARGF14
MOVJ C00106 BC00106 VJ=20.00  +MOVJ EC00106 VJ=20.00
SFTON3D P023
SMOVL C00107 BC00107 V=133.3  +MOVJ EC00107
ARCON
SMOVL C00108 BC00108 V=10.0  +MOVJ EC00108
SMOVL C00109 BC00109 V=10.0  +MOVJ EC00109
ARCOF
SFTOF3D
MOVJ C00110 BC00110 VJ=15.00  +MOVJ EC00110 VJ=15.00
MOVJ C00111 BC00111 VJ=100.00  +MOVJ EC00111 VJ=15.00
MOVJ C00112 BC00112 VJ=100.00  +MOVJ EC00112 VJ=100.00
SFTON3D P022
SMOVL C00113 BC00113 V=83.3  +MOVJ EC00113
ARCON
SMOVL C00114 BC00114 V=9.2  +MOVJ EC00114
SMOVL C00115 BC00115 V=9.2  +MOVJ EC00115
SMOVL C00116 BC00116 V=11.7  +MOVJ EC00116
SMOVL C00117 BC00117 V=11.7  +MOVJ EC00117
SMOVL C00118 BC00118 V=11.7  +MOVJ EC00118
SMOVL C00119 BC00119 V=11.7  +MOVJ EC00119
SMOVC C00120 BC00120 V=10.0  +MOVJ EC00120
SMOVC C00121 BC00121 V=10.0  +MOVJ EC00121
SMOVC C00122 BC00122 V=10.0  +MOVJ EC00122
SMOVL C00123 BC00123 V=10.0  +MOVJ EC00123
ARCOF
SFTOF3D
MOVJ C00124 BC00124 VJ=15.00  +MOVJ EC00124 VJ=15.00
MOVJ C00125 BC00125 VJ=40.00  +MOVJ EC00125 VJ=15.00
MACRO1 MJ#(0) ARGF6
SFTON3D P021
MOVJ C00126 BC00126 VJ=100.00  +MOVJ EC00126 VJ=40.00
SMOVL C00127 BC00127 V=250.0  +MOVJ EC00127
ARCON
SMOVL C00128 BC00128 V=8.3  +MOVJ EC00128
ARCOF
MOVJ C00129 BC00129 VJ=100.00  +MOVJ EC00129 VJ=100.00
SFTOF3D
MOVJ C00130 BC00130 VJ=100.00  +MOVJ EC00130 VJ=100.00
MOVJ C00131 BC00131 VJ=100.00  +MOVJ EC00131 VJ=100.00
MOVJ C00132 BC00132 VJ=100.00  +MOVJ EC00132 VJ=100.00
SMOVL C00133 BC00133 V=1000.0  +MOVJ EC00133
SFTON3D P071
SMOVL C00134 BC00134 V=400.0  +MOVJ EC00134
SMOVL C00135 BC00135 V=166.7  +MOVJ EC00135
SMOVL C00136 BC00136 V=100.0 PL=0  +MOVJ EC00136
MACRO1 MJ#(0) ARGF9
ARCON
SMOVL C00137 BC00137 V=6.7  +MOVJ EC00137
SWVON WEV#(205)
SMOVL C00138 BC00138 V=6.7  +MOVJ EC00138
ARCOF
SWVOF
SMOVL C00139 BC00139 V=100.0  +MOVJ EC00139
SMOVL C00140 BC00140 V=100.0  +MOVJ EC00140
TIMER T=5.00
SMOVL C00141 BC00141 V=100.0 PL=0  +MOVJ EC00141
SWVON WEV#(205)
ARCON
SMOVL C00142 BC00142 V=5.0  +MOVJ EC00142
ARCOF
SWVOF
SFTOF3D
SMOVL C00143 BC00143 V=400.0  +MOVJ EC00143
SMOVL C00144 BC00144 V=1000.0  +MOVJ EC00144
MOVJ C00145 BC00145 VJ=100.00  +MOVJ EC00145 VJ=100.00
CALL JOB:CLEAN-R1_KM_NEW
MOVJ C00146 BC00146 VJ=100.00  +MOVJ EC00146 VJ=100.00
SFTOF3D
MOVJ C00147 BC00147 VJ=100.00  +MOVJ EC00147 VJ=100.00
MOVJ C00148 BC00148 VJ=100.00  +MOVJ EC00148 VJ=100.00
MOVJ C00149 BC00149 VJ=100.00  +MOVJ EC00149 VJ=100.00
SMOVL C00150 BC00150 V=100.0  +MOVJ EC00150
SREFP 3 C00151 BC00151  +REFP EC00151
CALL JOB:SEARCH-R1-S13D
SET P021 P006
SFTON3D P021
SMOVL C00152 BC00152 V=100.0  +MOVJ EC00152
SREFP 3 C00153 BC00153  +REFP EC00153
CALL JOB:SEARCH-R1-S13D
SET P021 P006
SFTON3D P021
SMOVL C00154 BC00154 V=100.0  +MOVJ EC00154
SFTOF3D
SMOVL C00155 BC00155 V=250.0  +MOVJ EC00155
SMOVL C00156 BC00156 V=100.0  +MOVJ EC00156
SREFP 3 C00157 BC00157  +REFP EC00157
CALL JOB:SEARCH-R1-S13D
SET P022 P006
SFTON3D P022
SMOVL C00158 BC00158 V=100.0  +MOVJ EC00158
SREFP 3 C00159 BC00159  +REFP EC00159
CALL JOB:SEARCH-R1-S13D
SET P022 P006
SFTON3D P022
SMOVL C00160 BC00160 V=100.0  +MOVJ EC00160
SFTOF3D
MOVJ C00161 BC00161 VJ=100.00  +MOVJ EC00161 VJ=100.00
MOVJ C00162 BC00162 VJ=100.00  +MOVJ EC00162 VJ=100.00
MOVJ C00163 BC00163 VJ=100.00  +MOVJ EC00163 VJ=100.00
SMOVL C00164 BC00164 V=100.0  +MOVJ EC00164
SREFP 3 C00165 BC00165  +REFP EC00165
CALL JOB:SEARCH-R1-S13D
SET P023 P006
SFTON3D P023
SMOVL C00166 BC00166 V=100.0  +MOVJ EC00166
SREFP 3 C00167 BC00167  +REFP EC00167
CALL JOB:SEARCH-R1-S13D
SET P023 P006
SFTON3D P023
SMOVL C00168 BC00168 V=100.0  +MOVJ EC00168
SFTOF3D
MOVL C00169 BC00169 V=333.3  +MOVJ EC00169 VJ=100.00
SMOVL C00170 BC00170 V=100.0  +MOVJ EC00170
SREFP 3 C00171 BC00171  +REFP EC00171
CALL JOB:SEARCH-R1-S13D
SET P024 P006
SFTON3D P024
SMOVL C00172 BC00172 V=100.0  +MOVJ EC00172
SREFP 3 C00173 BC00173  +REFP EC00173
CALL JOB:SEARCH-R1-S13D
SET P024 P006
SFTON3D P024
SMOVL C00174 BC00174 V=100.0  +MOVJ EC00174
MOVJ C00175 BC00175 VJ=100.00  +MOVJ EC00175 VJ=100.00
MOVJ C00176 BC00176 VJ=100.00  +MOVJ EC00176 VJ=100.00
MOVJ C00177 BC00177 VJ=100.00  +MOVJ EC00177 VJ=100.00
MOVJ C00178 BC00178 VJ=100.00  +MOVJ EC00178 VJ=100.00
MOVJ C00179 BC00179 VJ=100.00  +MOVJ EC00179 VJ=100.00
SMOVL C00180 BC00180 V=100.0  +MOVJ EC00180
SREFP 3 C00181 BC00181  +REFP EC00181
CALL JOB:SEARCH-R1-S13D
SET P030 P006
SFTON3D P030
SMOVL C00182 BC00182 V=100.0  +MOVJ EC00182
SREFP 3 C00183 BC00183  +REFP EC00183
CALL JOB:SEARCH-R1-S13D
SET P030 P006
SFTON3D P030
SMOVL C00184 BC00184 V=100.0  +MOVJ EC00184
SMOVL C00185 BC00185 V=100.0  +MOVJ EC00185
SREFP 3 C00186 BC00186  +REFP EC00186
CALL JOB:SEARCH-R1-S13D
SET P030 P006
SFTON3D P030
SMOVL C00187 BC00187 V=100.0  +MOVJ EC00187
SFTOF3D
MOVJ C00188 BC00188 VJ=100.00  +MOVJ EC00188 VJ=100.00
MOVJ C00189 BC00189 VJ=100.00  +MOVJ EC00189 VJ=100.00
SMOVL C00190 BC00190 V=100.0  +MOVJ EC00190
SREFP 3 C00191 BC00191  +REFP EC00191
CALL JOB:SEARCH-R1-S13D
SET P031 P006
SFTON3D P031
SMOVL C00192 BC00192 V=100.0  +MOVJ EC00192
SREFP 3 C00193 BC00193  +REFP EC00193
CALL JOB:SEARCH-R1-S13D
SET P031 P006
SFTON3D P031
SMOVL C00194 BC00194 V=100.0  +MOVJ EC00194
SFTOF3D
MOVL C00195 BC00195 V=333.3  +MOVJ EC00195 VJ=100.00
SMOVL C00196 BC00196 V=100.0  +MOVJ EC00196
SREFP 3 C00197 BC00197  +REFP EC00197
CALL JOB:SEARCH-R1-S13D
SET P032 P006
SFTON3D P032
SMOVL C00198 BC00198 V=100.0  +MOVJ EC00198
SREFP 3 C00199 BC00199  +REFP EC00199
CALL JOB:SEARCH-R1-S13D
SET P032 P006
SFTON3D P032
SMOVL C00200 BC00200 V=100.0  +MOVJ EC00200
SFTOF3D
MOVJ C00201 BC00201 VJ=100.00  +MOVJ EC00201 VJ=100.00
MOVJ C00202 BC00202 VJ=100.00  +MOVJ EC00202 VJ=100.00
MOVJ C00203 BC00203 VJ=100.00  +MOVJ EC00203 VJ=100.00
MOVJ C00204 BC00204 VJ=100.00  +MOVJ EC00204 VJ=100.00
MOVJ C00205 BC00205 VJ=100.00  +MOVJ EC00205 VJ=100.00
MOVL C00206 BC00206 V=333.3  +MOVJ EC00206 VJ=100.00
SMOVL C00207 BC00207 V=100.0  +MOVJ EC00207
SREFP 3 C00208 BC00208  +REFP EC00208
CALL JOB:SEARCH-R1-S13D
SET P072 P006
SFTON3D P072
SMOVL C00209 BC00209 V=100.0  +MOVJ EC00209
SMOVL C00210 BC00210 V=100.0  +MOVJ EC00210
SMOVL C00211 BC00211 V=100.0  +MOVJ EC00211
SREFP 3 C00212 BC00212  +REFP EC00212
CALL JOB:SEARCH-R1-S13D
SET P072 P006
SFTON3D P072
SMOVL C00213 BC00213 V=100.0  +MOVJ EC00213
SFTOF3D
SMOVL C00214 BC00214 V=1000.0  +MOVJ EC00214
MOVJ C00215 BC00215 VJ=100.00  +MOVJ EC00215 VJ=100.00
MOVJ C00216 BC00216 VJ=100.00  +MOVJ EC00216 VJ=100.00
SMOVL C00217 BC00217 V=100.0  +MOVJ EC00217
SREFP 3 C00218 BC00218  +REFP EC00218
CALL JOB:SEARCH-R1-S13D
SET P025 P006
SFTON3D P025
SMOVL C00219 BC00219 V=100.0  +MOVJ EC00219
SREFP 3 C00220 BC00220  +REFP EC00220
CALL JOB:SEARCH-R1-S13D
SET P025 P006
SFTON3D P025
SMOVL C00221 BC00221 V=100.0  +MOVJ EC00221
SMOVL C00222 BC00222 V=100.0  +MOVJ EC00222
SREFP 3 C00223 BC00223  +REFP EC00223
CALL JOB:SEARCH-R1-S13D
SET P025 P006
SFTON3D P025
SMOVL C00224 BC00224 V=100.0  +MOVJ EC00224
MOVJ C00225 BC00225 VJ=100.00  +MOVJ EC00225 VJ=100.00
MOVJ C00226 BC00226 VJ=100.00  +MOVJ EC00226 VJ=100.00
MOVJ C00227 BC00227 VJ=100.00  +MOVJ EC00227 VJ=100.00
SMOVL C00228 BC00228 V=100.0  +MOVJ EC00228
SREFP 3 C00229 BC00229  +REFP EC00229
CALL JOB:SEARCH-R1-S13D
SET P026 P006
SFTON3D P026
SMOVL C00230 BC00230 V=100.0  +MOVJ EC00230
SREFP 3 C00231 BC00231  +REFP EC00231
CALL JOB:SEARCH-R1-S13D
SET P026 P006
SFTON3D P026
SMOVL C00232 BC00232 V=100.0  +MOVJ EC00232
SMOVL C00233 BC00233 V=100.0  +MOVJ EC00233
SREFP 3 C00234 BC00234  +REFP EC00234
CALL JOB:SEARCH-R1-S13D
SET P026 P006
SFTON3D P026
SMOVL C00235 BC00235 V=100.0  +MOVJ EC00235
MOVJ C00236 BC00236 VJ=100.00  +MOVJ EC00236 VJ=100.00
MOVJ C00237 BC00237 VJ=100.00  +MOVJ EC00237 VJ=100.00
MOVJ C00238 BC00238 VJ=100.00  +MOVJ EC00238 VJ=100.00
SMOVL C00239 BC00239 V=100.0  +MOVJ EC00239
SREFP 3 C00240 BC00240  +REFP EC00240
CALL JOB:SEARCH-R1-S13D
SET P027 P006
SFTON3D P027
SMOVL C00241 BC00241 V=100.0  +MOVJ EC00241
SMOVL C00242 BC00242 V=100.0  +MOVJ EC00242
SMOVL C00243 BC00243 V=100.0  +MOVJ EC00243
SREFP 3 C00244 BC00244  +REFP EC00244
CALL JOB:SEARCH-R1-S13D
SET P027 P006
SFTON3D P027
SMOVL C00245 BC00245 V=100.0  +MOVJ EC00245
SREFP 3 C00246 BC00246  +REFP EC00246
CALL JOB:SEARCH-R1-S13D
SET P027 P006
SFTON3D P027
SMOVL C00247 BC00247 V=100.0  +MOVJ EC00247
MOVL C00248 BC00248 V=100.0  +MOVJ EC00248 VJ=100.00
MOVJ C00249 BC00249 VJ=100.00  +MOVJ EC00249 VJ=100.00
SMOVL C00250 BC00250 V=100.0  +MOVJ EC00250
SREFP 3 C00251 BC00251  +REFP EC00251
CALL JOB:SEARCH-R1-S13D
SET P028 P006
SFTON3D P028
SMOVL C00252 BC00252 V=100.0  +MOVJ EC00252
SMOVL C00253 BC00253 V=100.0  +MOVJ EC00253
SREFP 3 C00254 BC00254  +REFP EC00254
CALL JOB:SEARCH-R1-S13D
SET P028 P006
SFTON3D P028
SMOVL C00255 BC00255 V=100.0  +MOVJ EC00255
SMOVL C00256 BC00256 V=100.0  +MOVJ EC00256
SREFP 3 C00257 BC00257  +REFP EC00257
CALL JOB:SEARCH-R1-S13D
SET P028 P006
SFTON3D P028
SMOVL C00258 BC00258 V=100.0  +MOVJ EC00258
MOVJ C00259 BC00259 VJ=100.00  +MOVJ EC00259 VJ=100.00
MOVJ C00260 BC00260 VJ=100.00  +MOVJ EC00260 VJ=100.00
MOVJ C00261 BC00261 VJ=100.00  +MOVJ EC00261 VJ=100.00
MACRO1 MJ#(0) ARGF14
SMOVL C00262 BC00262 V=133.3  +MOVJ EC00262
ARCON
SMOVL C00263 BC00263 V=10.0  +MOVJ EC00263
ARCOF
MOVJ C00264 BC00264 VJ=100.00  +MOVJ EC00264 VJ=100.00
SFTOF3D
MOVJ C00265 BC00265 VJ=100.00  +MOVJ EC00265 VJ=100.00
MOVJ C00266 BC00266 VJ=100.00  +MOVJ EC00266 VJ=100.00
SFTON3D P027
SMOVL C00267 BC00267 V=133.3  +MOVJ EC00267
ARCON
SMOVL C00268 BC00268 V=10.0  +MOVJ EC00268
SMOVL C00269 BC00269 V=10.0  +MOVJ EC00269
SMOVL C00270 BC00270 V=10.8  +MOVJ EC00270
SMOVL C00271 BC00271 V=11.7  +MOVJ EC00271
SMOVC C00272 BC00272 V=11.7  +MOVJ EC00272
SMOVC C00273 BC00273 V=10.0  +MOVJ EC00273
SMOVC C00274 BC00274 V=10.0  +MOVJ EC00274
SMOVL C00275 BC00275 V=10.0  +MOVJ EC00275
ARCOF
MOVJ C00276 BC00276 VJ=100.00  +MOVJ EC00276 VJ=100.00
MOVJ C00277 BC00277 VJ=100.00  +MOVJ EC00277 VJ=100.00
SFTOF3D
MOVJ C00278 BC00278 VJ=100.00  +MOVJ EC00278 VJ=100.00
SFTON3D P026
SMOVL C00279 BC00279 V=133.3  +MOVJ EC00279
ARCON
SMOVL C00280 BC00280 V=10.0  +MOVJ EC00280
SMOVL C00281 BC00281 V=10.0  +MOVJ EC00281
SMOVL C00282 BC00282 V=10.0  +MOVJ EC00282
SMOVL C00283 BC00283 V=10.0  +MOVJ EC00283
ARCOF
MOVJ C00284 BC00284 VJ=100.00  +MOVJ EC00284 VJ=100.00
MOVJ C00285 BC00285 VJ=100.00  +MOVJ EC00285 VJ=100.00
SFTON3D P025
MOVJ C00286 BC00286 VJ=100.00  +MOVJ EC00286 VJ=100.00
MACRO1 MJ#(0) ARGF6
SMOVL C00287 BC00287 V=133.3  +MOVJ EC00287
ARCON
SMOVL C00288 BC00288 V=10.0  +MOVJ EC00288
SMOVL C00289 BC00289 V=10.0  +MOVJ EC00289
SMOVL C00290 BC00290 V=10.0  +MOVJ EC00290
SMOVL C00291 BC00291 V=10.0  +MOVJ EC00291
SMOVL C00292 BC00292 V=10.0  +MOVJ EC00292
ARCOF
SFTOF3D
MOVJ C00293 BC00293 VJ=100.00  +MOVJ EC00293 VJ=100.00
MOVJ C00294 BC00294 VJ=100.00  +MOVJ EC00294 VJ=100.00
MOVJ C00295 BC00295 VJ=100.00  +MOVJ EC00295 VJ=100.00
MOVJ C00296 BC00296 VJ=100.00  +MOVJ EC00296 VJ=100.00
SMOVL C00297 BC00297 V=166.7  +MOVJ EC00297
SFTON3D P072
SMOVL C00298 BC00298 V=100.0 PL=0  +MOVJ EC00298
MACRO1 MJ#(0) ARGF9
ARCON
SMOVL C00299 BC00299 V=6.7  +MOVJ EC00299
SWVON WEV#(205)
SMOVL C00300 BC00300 V=6.7  +MOVJ EC00300
ARCOF
SWVOF
SMOVL C00301 BC00301 V=166.7  +MOVJ EC00301
SMOVL C00302 BC00302 V=166.7  +MOVJ EC00302
TIMER T=5.00
SMOVL C00303 BC00303 V=100.0 PL=0  +MOVJ EC00303
ARCON
SWVON WEV#(205)
SMOVL C00304 BC00304 V=5.0  +MOVJ EC00304
ARCOF
SWVOF
SMOVL C00305 BC00305 V=166.7  +MOVJ EC00305
SFTOF3D
MOVL C00306 BC00306 V=1000.0  +MOVJ EC00306 VJ=100.00
MOVJ C00307 BC00307 VJ=100.00  +MOVJ EC00307 VJ=100.00
MOVJ C00308 BC00308 VJ=100.00  +MOVJ EC00308 VJ=100.00
MOVJ C00309 BC00309 VJ=100.00  +MOVJ EC00309 VJ=100.00
MOVJ C00310 BC00310 VJ=100.00  +MOVJ EC00310 VJ=100.00
MACRO1 MJ#(0) ARGF14
MOVJ C00311 BC00311 VJ=100.00  +MOVJ EC00311 VJ=100.00
SFTON3D P023
SMOVL C00312 BC00312 V=133.3  +MOVJ EC00312
ARCON
SWVON WEV#(14)
SFTON3D P024
SMOVL C00313 BC00313 V=7.5  +MOVJ EC00313
ARCOF
SWVOF
MOVJ C00314 BC00314 VJ=100.00  +MOVJ EC00314 VJ=100.00
MOVJ C00315 BC00315 VJ=100.00  +MOVJ EC00315 VJ=100.00
MOVJ C00316 BC00316 VJ=100.00  +MOVJ EC00316 VJ=100.00
MOVJ C00317 BC00317 VJ=100.00  +MOVJ EC00317 VJ=100.00
SFTON3D P021
SMOVL C00318 BC00318 V=133.3  +MOVJ EC00318
SREFP 1 C00319 BC00319  +REFP EC00319
SREFP 2 C00320 BC00320  +REFP EC00320
ARCON
SWVON WEV#(14)
SFTON3D P022
SMOVL C00321 BC00321 V=7.5  +MOVJ EC00321
ARCOF
SWVOF
MOVJ C00322 BC00322 VJ=100.00  +MOVJ EC00322 VJ=100.00
MOVJ C00323 BC00323 VJ=100.00  +MOVJ EC00323 VJ=100.00
MOVJ C00324 BC00324 VJ=100.00  +MOVJ EC00324 VJ=100.00
MOVJ C00325 BC00325 VJ=100.00  +MOVJ EC00325 VJ=100.00
MOVJ C00326 BC00326 VJ=100.00  +MOVJ EC00326 VJ=100.00
MOVJ C00327 BC00327 VJ=100.00  +MOVJ EC00327 VJ=100.00
MOVJ C00328 BC00328 VJ=100.00  +MOVJ EC00328 VJ=100.00
MACRO1 MJ#(0) ARGF9
SFTON3D P030
SMOVL C00329 BC00329 V=133.3 PL=0  +MOVJ EC00329
SREFP 1 C00330 BC00330  +REFP EC00330
SREFP 2 C00331 BC00331  +REFP EC00331
SWVON WEV#(68)
ARCON
SMOVL C00332 BC00332 V=10.0  +MOVJ EC00332
SMOVL C00333 BC00333 V=10.0  +MOVJ EC00333
SMOVL C00334 BC00334 V=10.0  +MOVJ EC00334
COMM SMOVL C00335 BC00335 V=10.0  +MOVJ EC00335
ARCOF
SWVOF
MOVJ C00336 BC00336 VJ=100.00  +MOVJ EC00336 VJ=100.00
MOVJ C00337 BC00337 VJ=100.00  +MOVJ EC00337 VJ=100.00
SMOVL C00338 BC00338 V=133.3 PL=0  +MOVJ EC00338
ARCON
SWVON WEV#(61)
SMOVL C00339 BC00339 V=8.3  +MOVJ EC00339
ARCOF
SWVOF
MOVJ C00340 BC00340 VJ=100.00  +MOVJ EC00340 VJ=100.00
MOVJ C00341 BC00341 VJ=100.00  +MOVJ EC00341 VJ=100.00
SFTON3D P032
MOVJ C00342 BC00342 VJ=100.00  +MOVJ EC00342 VJ=100.00
MACRO1 MJ#(0) ARGF9
SMOVL C00343 BC00343 V=133.3  +MOVJ EC00343
ARCON
SMOVL C00344 BC00344 V=8.3  +MOVJ EC00344
SFTON3D P031
SWVON WEV#(61)
SMOVL C00345 BC00345 V=10.0  +MOVJ EC00345
SMOVL C00346 BC00346 V=10.0  +MOVJ EC00346
SMOVL C00347 BC00347 V=10.0  +MOVJ EC00347
ARCOF
SWVOF
MOVJ C00348 BC00348 VJ=100.00  +MOVJ EC00348 VJ=100.00
SFTOF3D
MOVJ C00349 BC00349 VJ=100.00  +MOVJ EC00349 VJ=100.00
MOVJ C00350 BC00350 VJ=100.00  +MOVJ EC00350 VJ=100.00
MOVJ C00351 BC00351 VJ=100.00  +MOVJ EC00351 VJ=100.00
MOVJ C00352 BC00352 VJ=100.00  +MOVJ EC00352 VJ=100.00
MOVJ C00353 BC00353 VJ=100.00  +MOVJ EC00353 VJ=100.00
MOVJ C00354 BC00354 VJ=100.00  +MOVJ EC00354 VJ=100.00
MOVJ C00355 BC00355 VJ=100.00  +MOVJ EC00355 VJ=100.00
MACRO1 MJ#(0) ARGF9
SFTON3D P023
SMOVL C00356 BC00356 V=133.3  +MOVJ EC00356
SREFP 2 C00357 BC00357  +REFP EC00357
SREFP 1 C00358 BC00358  +REFP EC00358
ARCON
SWVON WEV#(14)
SMOVL C00359 BC00359 V=8.3  +MOVJ EC00359
ARCOF
SWVOF
MOVJ C00360 BC00360 VJ=100.00  +MOVJ EC00360 VJ=100.00
MOVJ C00361 BC00361 VJ=100.00  +MOVJ EC00361 VJ=100.00
SFTON3D P021
SMOVL C00362 BC00362 V=133.3  +MOVJ EC00362
ARCON
SWVON WEV#(14)
SMOVL C00363 BC00363 V=8.3  +MOVJ EC00363
ARCOF
SWVOF
SFTOF3D
MOVJ C00364 BC00364 VJ=100.00  +MOVJ EC00364 VJ=100.00
MOVJ C00365 BC00365 VJ=100.00  +MOVJ EC00365 VJ=100.00
MOVJ C00366 BC00366 VJ=100.00  +MOVJ EC00366 VJ=100.00
MOVJ C00367 BC00367 VJ=100.00  +MOVJ EC00367 VJ=100.00
MOVJ C00368 BC00368 VJ=100.00  +MOVJ EC00368 VJ=100.00
MOVJ C00369 BC00369 VJ=100.00  +MOVJ EC00369 VJ=100.00
'KONIEC
END
